Yaskawa INFORM job: R1_W43-44-A2(80,180)KM-OK_MOD.JBI

/JOB
//NAME R1_W43-44-A2(80,180)KM-OK_MOD
///FOLDERNAME KRIS-SCIANA
//POS
///NPOS 92,92,0,2,0,0
///TOOL 0
///POSTYPE PULSE
///PULSE
C00000=-1999,180198,107788,-13936,86373,83899
C00001=-1999,180198,107788,-13936,86373,83899
C00002=-43273,105049,47365,-19266,82618,17073
C00003=-71921,52889,5426,-22965,80012,32608
C00004=-125539,-44737,-73069,-29889,75135,61684
C00005=-128409,-43805,-69644,-28832,72769,61239
C00006=-129164,-43691,-67457,-28680,71391,61311
C00007=-129516,-43610,-67407,-28519,71287,61204
C00008=-128716,-43399,-68593,-28756,72284,61249
C00009=-125452,-43071,-69586,-30042,74080,61968
C00010=-130187,-11295,-57221,-29955,89458,59830
C00011=-137590,-27816,-65842,-19359,69291,63411
C00012=-137552,-28488,-64323,-19538,68090,63627
C00013=-137425,-28335,-61936,-19796,66808,63895
C00014=-137563,-29297,-63389,-19663,67152,63785
C00015=-138865,-39574,-72842,-18843,67381,63290
C00016=-136116,-57579,-72593,-22873,56489,58406
C00017=-136116,-57656,-72199,-22944,56229,58465
C00018=-136116,-57579,-72593,-22873,56489,58406
C00019=-135007,-59068,-74434,-23478,57129,58722
C00020=-132124,-62672,-78933,-25018,58781,59524
C00021=-120651,-21229,-57646,-40322,87510,70819
C00022=-123210,-22722,-55716,-39523,84917,70774
C00023=-124330,-23596,-55696,-39169,84087,70633
C00024=-124217,-22317,-55487,-39184,84548,70508
C00025=-123155,-23314,-54934,-39574,84326,71016
C00026=-124227,-19270,-52147,-39202,84158,70648
C00027=-123139,-18387,-52130,-39545,84963,70786
C00028=-120649,-16917,-54042,-40323,87510,70820
C00029=-116125,-44661,-62928,-56166,74056,-59527
C00030=-118631,-43374,-59008,-55785,71602,-59330
C00031=-119697,-42424,-57655,-55534,70789,-59407
C00032=-118663,-44204,-58389,-55988,71116,-59017
C00033=-119609,-42204,-58263,-55432,71123,-59582
C00034=-121132,-46387,-60546,-55138,69808,-59596
C00035=-127786,-52615,-64375,-50280,62099,-62151
C00036=-117551,-45324,-73752,-54437,76971,-62238
C00037=-117551,-45324,-73752,-54437,76971,-62238
C00038=-161657,-30726,-79920,772,93057,-50157
C00039=-181669,-13323,-64922,23952,108211,-55227
C00040=-180420,-18454,-65224,23348,105655,-55351
C00041=-179762,-19978,-65109,23091,104712,-55325
C00042=-180997,-20082,-65170,23353,104994,-55678
C00043=-179767,-19299,-65754,23201,105398,-55188
C00044=-180772,-17933,-63381,23309,104943,-55615
C00045=-178692,-14024,-59763,22865,104235,-55070
C00046=-181365,-16668,-63571,23526,105793,-55635
C00047=-157540,-55913,-92611,1182,92318,-32543
C00048=-155778,-26705,-72811,-3028,103995,-32959
C00049=-155015,-27488,-73346,-3191,103948,-32728
C00050=-154801,-27902,-73351,-3233,103746,-32658
C00051=-151236,-37378,-85109,-9837,103355,-33029
C00052=-163460,-35194,-90423,20298,108366,-49466
C00053=-147151,-121982,-123348,-5805,52349,-43157
C00054=-27981,-121982,-123348,-5805,52349,-43157
C00055=-64129,-68336,-105858,8437,79945,-45520
C00056=-77063,-8149,-55226,12189,87021,-43056
C00057=-57716,14735,-27514,-8279,72578,-25222
C00058=-58232,14892,-24839,-8078,70982,-25281
C00059=-58063,17340,-22233,-8185,70657,-25202
C00060=-58472,15435,-24293,-7956,70902,-25355
C00061=-59491,14531,-24173,-7445,70279,-25652
C00062=-57194,14795,-23002,-8680,69914,-24859
C00063=-57174,14609,-22764,-8703,69675,-24835
C00064=-57683,13071,-24957,-8407,70177,-25044
C00065=-56826,12123,-28333,-8777,71835,-24880
C00066=-51865,34324,-22123,-10735,79789,64704
C00067=-59101,8612,-35422,3885,58670,66532
C00068=-63108,16408,-20626,7237,53846,64801
C00069=-63816,18405,-18773,7796,53795,64519
C00070=-62681,15567,-23734,6783,55283,65059
C00071=-58140,26959,-12922,3339,54223,66731
C00072=-58524,28773,-8935,3705,52721,66532
C00073=-59265,30460,-7226,4300,52573,66235
C00074=-58187,22167,-20055,3299,56150,66776
C00075=-55114,35104,-14749,-11639,72465,63679
C00076=-59261,25940,-16255,-4057,60712,64739
C00077=-54858,38521,-3460,-7130,59593,66369
C00078=-47704,48120,-9634,-15389,76990,65485
C00079=-46882,45180,-4962,-16115,72902,66280
C00080=-47835,37934,-3746,-16016,68426,66575
C00081=-50553,27764,-14014,-14439,69013,65563
C00082=-50621,26831,-15159,-14384,69226,65512
C00083=-50869,27036,-14182,-14292,68705,65492
C00084=-50998,26612,-14598,-14219,68722,65446
C00085=-51149,26075,-14744,-14152,68515,65416
C00086=-49257,22630,-27080,-14715,74460,65315
C00087=-56826,24849,-38650,-8422,84586,-25767
C00088=-78114,-99903,-117821,2511,49690,-31810
C00089=-78114,-99903,-117821,2511,30862,-31810
C00090=3198,-156648,-132716,2511,-14356,-31810
C00091=3198,-156648,-132716,2511,-14356,-31810
BC00000=82357,1835,1075208
BC00001=241769,1835,1075208
BC00002=294022,1227,1075197
BC00003=389321,805,1075189
BC00004=398174,15,1075175
BC00005=398174,15,1075175
BC00006=398174,15,1075175
BC00007=398174,15,1075175
BC00008=398174,15,1075175
BC00009=398174,15,1075175
BC00010=398174,15,1075175
BC00011=398174,15,1075175
BC00012=398174,15,1075175
BC00013=398174,15,1075175
BC00014=398174,15,1075175
BC00015=398174,15,1075175
BC00016=398174,15,1075175
BC00017=398174,15,1075175
BC00018=398174,15,1075175
BC00019=398174,15,1075175
BC00020=398174,15,1075175
BC00021=398174,15,1075175
BC00022=398174,15,1075175
BC00023=398174,15,1075175
BC00024=398174,15,1075175
BC00025=398174,15,1075175
BC00026=398174,15,1075175
BC00027=398174,15,1075175
BC00028=398174,15,1075175
BC00029=398174,15,1075175
BC00030=398174,15,1075175
BC00031=398174,15,1075175
BC00032=398174,15,1075175
BC00033=398174,15,1075175
BC00034=398174,15,1075175
BC00035=398174,15,1075175
BC00036=398174,15,1075175
BC00037=398174,15,1075175
BC00038=398174,10899,1075175
BC00039=398174,25865,1075175
BC00040=398174,28772,1075175
BC00041=398174,29936,1075169
BC00042=398174,29935,1075175
BC00043=398174,29935,1075175
BC00044=398174,33387,1075175
BC00045=398174,33387,1075175
BC00046=398174,32225,1075175
BC00047=398174,32225,1075175
BC00048=398174,32225,1075175
BC00049=398174,32225,1075175
BC00050=398174,32225,1075175
BC00051=398174,32225,1075175
BC00052=398174,29318,1075175
BC00053=372318,14254,1052622
BC00054=185802,37675,1052622
BC00055=160909,26210,1065038
BC00056=140585,16850,1075175
BC00057=87282,15,1075175
BC00058=92863,15,1075175
BC00059=92863,15,1075175
BC00060=95096,15,1075175
BC00061=95096,15,1075175
BC00062=92863,15,1075175
BC00063=92863,15,1075175
BC00064=92830,15,1075175
BC00065=87249,15,1075175
BC00066=87249,15,1075175
BC00067=87249,15,1075175
BC00068=87249,15,1075175
BC00069=87249,15,1075175
BC00070=87249,15,1075175
BC00071=87249,15,1075175
BC00072=87249,15,1075175
BC00073=87249,15,1075175
BC00074=87249,15,1075175
BC00075=87249,15,1075175
BC00076=87249,15,1075175
BC00077=87249,15,1075175
BC00078=87249,15,1075175
BC00079=87249,15,1075175
BC00080=87249,15,1075175
BC00081=87249,15,1075175
BC00082=87249,15,1075174
BC00083=87249,15,1075174
BC00084=87249,15,1075174
BC00085=87249,15,1075174
BC00086=87249,15,1075174
BC00087=87249,15,1075175
BC00088=87249,15,1075175
BC00089=87249,15,1075175
BC00090=24328,15,1075175
BC00091=24328,497765,1075175
///POSTYPE BASE
///RECTAN
///RCONF 0,0,0,0,1,0,0,0,0,0,0,0,0,0,0,0,0,0,0,0,0,0,0,0
P00006=2.006,1.622,-0.565,0.0000,0.0000,0.0000
///RCONF 0,0,0,0,0,0,0,0,0,0,0,0,0,0,0,0,0,0,0,0,0,0,0,0
P00023=-2.957,-4.083,2.762,0.0000,0.0000,0.0000
//INST
///DATE 2025/01/20 11:10
///ATTR SC,RW
///GROUP1 RB1,BS1
NOP
'r1_W43-44-A2(80,180)
'Path S1263
SFTOF
MOVJ C00000 BC00000 VJ=100.00
MOVJ C00001 BC00001 VJ=100.00
MOVJ C00002 BC00002 VJ=100.00
MOVJ C00003 BC00003 VJ=100.00
MOVJ C00004 BC00004 VJ=100.00
MOVJ C00005 BC00005 VJ=20.00
MOVL C00006 BC00006 V=60.0
REFP 3 C00007 BC00007
CALL JOB:SEARCH-R1
SET P023 P006
SFTON P023
MOVL C00008 BC00008 V=60.0
MOVJ C00009 BC00009 VJ=20.00
MOVL C00010 BC00010 V=166.7
MOVL C00011 BC00011 V=166.7
MOVL C00012 BC00012 V=166.7
REFP 3 C00013 BC00013
CALL JOB:SEARCH-R1
SET P023 P006
SFTON P023
MOVL C00014 BC00014 V=166.7
MOVL C00015 BC00015 V=166.7
MOVL C00016 BC00016 V=166.7
REFP 3 C00017 BC00017
CALL JOB:SEARCH-R1
SET P023 P006
SFTON P023
MOVL C00018 BC00018 V=60.0
MOVL C00019 BC00019 V=166.7
MOVL C00020 BC00020 V=400.0
'Path W1265
SFTOF
SFTON P023
CALL JOB:COFNIJ_DRUT
MOVJ C00021 BC00021 VJ=20.00
MOVJ C00022 BC00022 VJ=20.00
MOVL C00023 BC00023 V=100.0 PL=0
REFP 1 C00024 BC00024
REFP 2 C00025 BC00025
MACRO1 MJ#(0) ARGF7
ARCON
MOVL C00026 BC00026 V=10.8
ARCOF
MOVL C00027 BC00027 V=100.0
MOVL C00028 BC00028 V=166.7
SFTOF
'Path W1266
SFTOF
SFTON P023
MOVJ C00029 BC00029 VJ=20.00
MOVJ C00030 BC00030 VJ=20.00
MOVL C00031 BC00031 V=100.0 PL=0
REFP 1 C00032 BC00032
REFP 2 C00033 BC00033
MACRO1 MJ#(0) ARGF7
ARCON
MOVL C00034 BC00034 V=10.8
MOVL C00035 BC00035 V=10.8
ARCOF
MOVL C00036 BC00036 V=100.0
MOVL C00037 BC00037 V=166.7
SFTOF
'Path W1268
SFTOF
MOVJ C00038 BC00038 VJ=20.00
'Path W1269
SFTOF
SFTON P023
MOVJ C00039 BC00039 VJ=20.00
MOVJ C00040 BC00040 VJ=20.00
MOVL C00041 BC00041 V=100.0 PL=0
REFP 1 C00042 BC00042
REFP 2 C00043 BC00043
MACRO1 MJ#(0) ARGF7
ARCON
MOVL C00044 BC00044 V=10.8
MOVL C00045 BC00045 V=10.8
ARCOF
MOVL C00046 BC00046 V=100.0
MOVL C00047 BC00047 V=166.7
MOVL C00048 BC00048 V=166.7 PL=0
ARCON
MOVL C00049 BC00049 V=10.0
MOVL C00050 BC00050 V=10.0
ARCOF
MOVL C00051 BC00051 V=166.7
SFTOF
'Path VIA1273
SFTOF
MOVJ C00052 BC00052 VJ=20.00
'Path VIA1274
SFTOF
MOVJ C00053 BC00053 VJ=20.00
'Path VIA1275
SFTOF
MOVJ C00054 BC00054 VJ=20.00
'Path W1270
SFTOF
SFTON P023
MOVJ C00055 BC00055 VJ=20.00
MOVJ C00056 BC00056 VJ=20.00
'Path W1271
SFTOF
SFTON P023
MOVJ C00057 BC00057 VJ=20.00
MOVJ C00058 BC00058 VJ=20.00
MOVL C00059 BC00059 V=100.0 PL=0
REFP 1 C00060 BC00060
REFP 2 C00061 BC00061
MACRO1 MJ#(0) ARGF7
ARCON
MOVL C00062 BC00062 V=10.0
MOVL C00063 BC00063 V=13.3
ARCOF
MOVL C00064 BC00064 V=100.0
MOVL C00065 BC00065 V=166.7
MOVJ C00066 BC00066 VJ=20.00
MOVJ C00067 BC00067 VJ=10.00
COMM MACRO1 MJ#(0) ARGF7
COMM MOVJ C00068 BC00068 VJ=10.00
COMM 'ARCON
COMM MOVL C00069 BC00069 V=10.8
COMM 'ARCOFF
COMM MOVJ C00070 BC00070 VJ=10.00
COMM MOVJ C00071 BC00071 VJ=10.00
COMM MACRO1 MJ#(0) ARGF6
COMM MOVJ C00072 BC00072 VJ=10.00
COMM 'ARCON
COMM MOVL C00073 BC00073 V=10.0
COMM 'ARCOFF
MOVJ C00074 BC00074 VJ=10.00
SFTOF
MOVJ C00075 BC00075 VJ=20.00
SFTON P023
MACRO1 MJ#(0) ARGF7
MOVJ C00076 BC00076 VJ=20.00 PL=0
ARCON
MOVL C00077 BC00077 V=7.5
ARCOF
MOVJ C00078 BC00078 VJ=20.00
MOVJ C00079 BC00079 VJ=10.00
MACRO1 MJ#(0) ARGF6
MOVJ C00080 BC00080 VJ=10.00
ARCON
TIMER T=0.20
ARCOF
MOVJ C00081 BC00081 VJ=10.00
ARCON
TIMER T=0.50
ARCOF
MOVJ C00082 BC00082 VJ=10.00
MOVL C00083 BC00083 V=100.0
ARCON
MOVL C00084 BC00084 V=5.0
MOVL C00085 BC00085 V=5.0
ARCOF
MOVJ C00086 BC00086 VJ=10.00
MOVJ C00087 BC00087 VJ=20.00
MOVJ C00088 BC00088 VJ=50.00
SFTOF
MOVJ C00089 BC00089 VJ=100.00
MOVJ C00090 BC00090 VJ=100.00
MOVJ C00091 BC00091 VJ=100.00
END
